FUNCTION_BLOCK FB_TMCM1140_Home
VAR_INPUT
	bExecute	: BOOL;
	bStop		: BOOL;
END_VAR
VAR_OUTPUT
	bBusy 		: BOOL;
	bError 		: BOOL;
	nErrorId 	: ERRORID;	
END_VAR
VAR_IN_OUT
	pHwRef : POINTER TO FB_HwRefTMCM1140;
END_VAR
VAR
	nState 			: USINT;
	nStateNext 		: USINT;
	bDigiout0 		: BOOL;
	bDigiout1 		: BOOL;
	fbSdoWrite 		: FB_SDO_WRITE;
	eCurrentHomingState : E_CoDS402HomingState;
END_VAR

IF bExecute THEN
	CASE nState OF
		0:	//Set Fast homing speed
			bBusy := TRUE;
			fbSdoWrite.nIndex := 16#6099;
			fbSdoWrite.nSubIndex := 1;
			fbSdoWrite.nDataLength := 4;
			fbSdoWrite.nData := pHwRef^.M_RealToInternSpeed(pHwRef^.P_nFastHomingSpeed);
			nState := 40;
			nStateNext := 1;
			
		1:	//Set Slow homing speed
			fbSdoWrite.nIndex := 16#6099;
			fbSdoWrite.nSubIndex := 2;
			fbSdoWrite.nDataLength := 4;
			fbSdoWrite.nData := pHwRef^.M_RealToInternSpeed(pHwRef^.P_nSlowHomingSpeed);
			nState := 40;
			nStateNext := 2;			

		2:	//Set homing methode
			fbSdoWrite.nIndex := 16#6098;
			fbSdoWrite.nSubIndex := 0;
			fbSdoWrite.nDataLength := 1;
			fbSdoWrite.nData := pHwRef^.P_eHomingMethode;
			nState := 40;
			nStateNext := 3;
			
		3: 	//Write home offset
			fbSdoWrite.nIndex := 16#607C;
			fbSdoWrite.nSubIndex := 0;
			fbSdoWrite.nDataLength := 4;
			fbSdoWrite.nData := pHwRef^.M_RealToInternPos(pHwRef^.P_nRefPos);
			nState := 40;
			nStateNext := 4;
			
		4:	//Write profile speed
			fbSdoWrite.nIndex := 16#6081;
			fbSdoWrite.nSubIndex := 0;
			fbSdoWrite.nDataLength := 4;
			fbSdoWrite.nData := pHwRef^.M_RealToInternSpeed(pHwRef^.P_nMaxSpeed);
			nState := 40;
			nStateNext := 5;

		5:	//Set Mode of operation to "6" (Homing)
			pHwRef^.nMode := 6; //Homing
			nState := 6;
			
		6:	//Start homing
			pHwRef^.nControlword := 31;
			nState := 7;
			
		7:	//Wait for State "Homing in process
			IF pHwRef^.M_GetDS402State() = E_CoDS402States.DS402STATE_OperationEnabled THEN
				IF bStop THEN
					pHwRef^.nControlword := 15;
					nState := 80;
				ELSE
					eCurrentHomingState := pHwRef^.M_GetHomingState();
					CASE eCurrentHomingState OF
						E_CoDS402HomingState.HomingAttainedButNotReached,
						E_CoDS402HomingState.HomingError,
						E_CoDS402HomingState.HomingInteruptedOrNotReached:
							nErrorId := E_ErrorIdDS402.ERRORID_HomingInterruptedOrNotReached;
							nState := 99;
						E_CoDS402HomingState.HomingSuccess:
							pHwRef^.nControlword := 15;
							pHwRef^.nMode := 1;	//PP mode
							pHwRef^.M_SetTargetPos(pHwRef^.P_nHomePos, FALSE);
							pHwRef^.P_bIsHomed := TRUE;
							nState := 8;
					END_CASE
				END_IF
			ELSE
				nErrorId := 43434;
				nState := 99;
			END_IF
			
		8:	//Move to HomePos
			pHwRef^.nControlword := 31;
			nState := 9;
			
		9:	//Wait for setpoint acknowledge
			IF pHwRef^.nStatusword.12 THEN
				pHwRef^.nControlword := 15;
				nState := 10;
			END_IF
			
		10:	//Wait for target reached
			IF pHwRef^.M_GetDS402State() = E_CoDS402States.DS402STATE_OperationEnabled THEN
				//Das HALT-Bit von von der TMCM1140 nicht unterstützt.
				//Man kann den Mode auf "0" setzen und dann sollter der Motor auch anhalten
				IF bStop THEN
					IF bStop THEN
						pHwRef^.nMode := 0;
						nState := 80;
					END_IF
				ELSE
					IF pHwRef^.nStatusword.10 THEN
						nState := 80;
					END_IF
				END_IF
			ELSE
				nErrorId := E_ErrorIdDS402.ERRORID_OperationNotEnabled;
				nState := 99;
			END_IF
			
	END_CASE
	
	//Sdo senden
	IF nState = 40 THEN
		fbSdoWrite(sADSNetID:= pHwRef^.P_sAdsNetId, nPortNr:= pHwRef^.P_nAdsPort, bExecute:= TRUE);
		IF NOT fbSdoWrite.bBusy THEN
			IF fbSdoWrite.bError THEN
				nErrorId := fbSdoWrite.nAdsErrorId;
				nState := 99;
			ELSE
				nState := nStateNext;
			END_IF
			fbSdoWrite(bExecute:= FALSE);
		END_IF		
	END_IF
	
	IF nState >= 80 THEN
		bBusy := FALSE;
		IF nState = 99 THEN
			bError := TRUE;
		END_IF
	END_IF

ELSE
	bBusy 	:= FALSE;
	bError 	:= FALSE;
	bStop 	:= FALSE;
	nState 	:= 0;
END_IF

END_FUNCTION_BLOCK

(* stored: Version 1.1.0.1, ProductVersion 3.1.4024.11
   POU FB_TMCM1140_Home: Id {59590c01-bf8c-45b7-b54f-93e38fd147c4}, SpecialFunc None *)
